// TIA Portal V20 export
TYPE "LKinCtrl_typeCOff3DPoint"
   STRUCT
      x : LReal;   // X
      y : LReal;   // Y
      z : LReal;   // Z
   END_STRUCT;
END_TYPE
